TYPE _00BE31_PLCTOHW_PDOS :
STRUCT
	
	outputByte_0 	 : BYTE;
	outputByte_1 	 : BYTE;

END_STRUCT
END_TYPE

(* stored: Version 1.1.0.1
   DUT _00BE31_PLCTOHW_PDOS: Id {4ee1009f-eada-4e3e-a7bc-f682737b636c} *)
